TYPE "PLCtoMES_MainCheckIn"
VERSION : 0.1
   STRUCT
      "P-PartIDReq" : Bool;
      "P-PartType" : String[28];
      "P-PartID" : Array[1..10] of String[48];
      "P-RecipeVer" : String[18];
      "P-DeviceID" : Int;
      "P-MoldID" : Int;
      Reserve : Array[1..443] of Byte;
   END_STRUCT;

END_TYPE

